	// ============ Common varaibles ==============================
	bAxisMoved						:		BOOL;						// History variable to save if axis has moved marker
	fbTriggerResetStart				:		R_TRIG;						// To diagnose rising edge of starting reset
	fbTriggerStartingStart			:		R_TRIG;						// To diagnose rising edge of starting start
END_VAR

// ===========================================================================
;
// ===========================================================================

PROPERTY bState_HaltDone : BOOL
GET
bState_HaltDone := bHaltDone;
END_GET
END_PROPERTY

PROPERTY bState_ResetDone : BOOL
GET
bState_ResetDone := bResetDone;
END_GET
END_PROPERTY

PROPERTY bState_StartingDone : BOOL
GET
bState_StartingDone := bStartingDone;
END_GET
END_PROPERTY

METHOD Enable
VAR_INPUT
	bComprAirEnable					:			BOOL;			// Enable of compressed air
	bAxisEnable						:			BOOL;			// Enable of axis
	bSensorEnable					:			BOOL;			// Enable of sensor
	bManualAxisEnable				:			BOOL;			// Enable manual axis control
END_VAR

VAR
	bManualEnable: BOOL;
END_VAR
	// Store inputs in local variables
	bCompresAirEnableLocal				:=				bComprAirEnable;
	bAxisEnableLocal					:=				bAxisEnable;
	bSensorEnableLocal					:=				bSensorEnable;
	bManualAxisEnableLocal				:=				bManualAxisEnable;
	
	// Axis enable
	fbAxis.Enable(bEnable				:=				bAxisEnableLocal);
	
	// Cylinder manual control enable 
	bManualCylinderEnableLocal			:=				bManualAxisEnableLocal		AND		bCompresAirEnableLocal;
	
	// Control buttons (enable Signal Handling)
	fbButtonAxisFw.Enable(bEnable		:=				bManualAxisEnableLocal		AND NOT fbButtonAxisBw.bOutputSignal);
	fbButtonAxisBw.Enable(bEnable		:=				bManualAxisEnableLocal		AND NOT fbButtonAxisFw.bOutputSignal);
END_METHOD

PROPERTY fAxisVelocity : LREAL
GET
fAxisVelocity := fAxisVelo;
END_GET
SET
fAxisVelo := fAxisVelocity;
END_SET
END_PROPERTY

METHOD Halt : BOOL
VAR_INPUT
	bHalt				:			BOOL;				// True if machine is in STATE ABORTING or STOPPING
END_VAR
	// Store halt request
	bHaltRequest				:=		bHalt;
	
	// Axis halt
	fbAxis.Halt(bDriveHalt		:=		bHaltRequest);
	
	// Setting halt state from axis feedback
	bHaltDone					:=		fbAxis.bState_HaltDone;
END_METHOD

METHOD InputOutput
VAR_INPUT
END_VAR
	// Axis buttons and output variables for axis
	fbButtonAxisFw.SetOutput();
	fbButtonAxisBw.SetOutput();

	bAxisError							:=					fbAxis.bError;
	nAxisErrorID						:=					fbAxis.nErrorID;
	bAxisMoves							:=					fbAxis.bMoving;
	
	fbButtonAxisFw.bInputSignal			:=					bButtonAxisFwIn;
	fbButtonAxisBw.bInputSignal			:=					bButtonAxisBwIn;
	bButtonAxisFwOut					:=					fbButtonAxisFw.bOutputSignal;
	bButtonAxisBwOut					:=					fbButtonAxisBw.bOutputSignal;
END_METHOD

METHOD Manual
VAR_INPUT
END_VAR

	IF fbButtonAxisFw.bOutputSignal THEN
		IF bHaltDone THEN
			bHaltDone	:=		FALSE;
		END_IF
		
		IF NOT bAxisMoved THEN
			bAxisMoved 	:=		TRUE;
		END_IF
		
		fbAxis.MoveFw();
		
	ELSIF fbButtonAxisBw.bOutputSignal THEN
		IF bHaltDone THEN
			bHaltDone	:=		FALSE;
		END_IF
		
		IF NOT bAxisMoved THEN
			bAxisMoved 	:=		TRUE;
		END_IF
	
		fbAxis.MoveBw();
	
	// No button is pressed and Halt is not done
	ELSIF NOT bHaltDone	THEN
		IF bAxisMoved THEN
			Halt(bHalt	:=	TRUE);
		END_IF
	
	// Halt done, but still requested
	ELSIF bHaltRequest THEN
		Halt(bHalt		:=	FALSE);
		
		bAxisMoved	:=	FALSE;
	END_IF
END_METHOD

METHOD Reset
VAR_INPUT
	bReset				:			BOOL;			// True if machine is in state RESETTING
END_VAR

	// Store reset request
	bResetRequest					:=			bReset;
	
	bAxisMoved						:=			FALSE;
	bHaltRequest					:=			FALSE;
	bHaltDone						:=			FALSE;
	
	// Trigger for resetting extending FBs 
	fbTriggerResetStart(CLK			:=			bReset);
	
	// Resetting axis
	fbAxis.Reset(bDriveReset		:=			bReset);
	
	bResetDone						:=			fbAxis.bState_ResetDone;
END_METHOD

METHOD Starting
VAR_INPUT
	bStarting					:				BOOL;			// True if machine is in state STARTING
END_VAR

	fbTriggerStartingStart(CLK			:=			bStarting);
	
	IF fbTriggerStartingStart.Q THEN
		bStartingDone					:=			FALSE;
	// Set axis velocity through axis property
		fbAxis.fTargetVelocity			:=			fAxisVelo;

	END_IF
	
	// Axis feedback from MC_Power of axis method Enable()
	IF fbAxis.bState_Enable THEN
		bStartingDone					:=			TRUE;
	END_IF
END_METHOD

METHOD Stop : BOOL
VAR_INPUT
	bStop					:				BOOL;				// True if machine is in state ABORTING or STOPPING
END_VAR
	// Store halt request
	bHaltRequest					:=				bStop;
	
	// Axis halt
	fbAxis.Stop(bDriveStop			:=				bHaltRequest);
	
	// Setting halt state from axis feedback
	bHaltDone						:=				fbAxis.bState_HaltDone;
END_METHOD

END_FUNCTION_BLOCK

// ---- 02_Subsystems/FB_SortingModule.TcPOU
FUNCTION_BLOCK FB_SortingModule EXTENDS FB_SubsystemRoot
VAR_INPUT
	bButtonCylMoveToWorkIn										:						BOOL;
	bButtonCylMoveToBaseIn										:						BOOL;
END_VAR
VAR_OUTPUT
	bCylError													:						BOOL;
	sCylErrorMsg												:						STRING;
	
	a_Temps														:						ARRAY [1..100] OF LREAL;
	
	bButtonCylMoveToWorkOut										:						BOOL;
	bButtonCylMoveToBaseOut										:						BOOL;
END_VAR
VAR
	bSorted														:						BOOL;								// Part picked at sorting module
	// Sensor with delay functionality
	fbSensorDelay												:						FB_SignalHandlingDelay;
	
	// Function block instance for cylinder
	fbCylinder													:						FB_CylinderBase;
	fbCylinderDiag												:						FB_CylinderDiag;
	fbCylinderTemp												:						FB_CylinderTemp;
	fbCylinderTempDiag											:						FB_CylinderTempDiag;
	fbCylinderTempRec											:						FB_CylinderTempRecord;
	// Interface instance for cylinder
	itfCylinder													:						I_Cylinder;
	// Time parameters for submodules
	tTimeOutCylinder											:						TIME;								// For cylinder with position diagnosis: time in which the cylinder shcould reach work / base position
	tTimeIntervalCylinder										:						TIME;								// Time of intervals to record the temperature of cylinder
	tSensorDelay												:						TIME;								// Sensor delay
	tMoveAxisDelay												:						TIME;								// Time delay to stop running axis
	// ========================== Temperature parameters for cylinder  ======================================================================
	nTempMinCyl													:						LREAL;								// For cylinder with temperature diagnosis: minimal temperature
	nTempMaxCyl													:						LREAL;								// For cylinder with temperature diagnosis: maximal temperature
	// Manual cylinder controll
	fbButtonCylMoveToWork										:						FB_SignalHandlingIntern;			// Button to move cylinder manually to work position
	fbButtonCylMoveToBase										:						FB_SignalHandlingIntern;			// Button to move cylinder manually to base position
	// Common variables
	fbTimerAxis													:						TON;								// Timer to run axis for certain amount of time
	fbTriggerCylAtWorkPos										:						R_TRIG;								// Trigger to recognize rising edge of cylinder being at work position
	eStateAutoAxis												:						E_StateSortingAutoAxis;				// State variable for automatic / semi-auto mode for axis movement
	eStateAutoCylinder											:						E_StateSortingAutoCylinder;			// State variable for automatic / semi-auto mode for cylinder movement
END_VAR

METHOD Automatic
VAR_INPUT
END_VAR
	fbTriggerCylAtWorkPos(		CLK			:=		itfCylinder.bState_AtWorkPos);

	CASE eStateAutoAxis OF
		
		E_StateSortingAutoAxis.WaitForCylinderAtWorkPos:
			IF fbTriggerCylAtWorkPos.Q THEN
				fbTimerAxis(	IN			:=		TRUE,
								PT			:=		tMoveAxisDelay);
				
				eStateAutoAxis				:=		E_StateSortingAutoAxis.MoveAxis;
			END_IF
		
		E_StateSortingAutoAxis.MoveAxis:
			fbTimerAxis();
			IF bHaltRequest THEN
				
				eStateAutoAxis				:=		E_StateSortingAutoAxis.StopAxis;
			ELSIF fbTimerAxis.Q THEN
				fbTimerAxis(	IN			:=		FALSE);
				
				bSorted						:=		TRUE;
			
				eStateAutoAxis				:=		E_StateSortingAutoAxis.StopAxis;
			ELSE
				fbAxis.MoveFw();
			END_IF
		
		E_StateSortingAutoAxis.StopAxis:
				bSorted						:=		FALSE;
				
				IF NOT bHaltDone THEN
					Stop(	bStop			:=		TRUE);
				ELSE	
					Stop(	bStop			:=		FALSE);
					eStateAutoAxis			:=		E_StateSortingAutoAxis.WaitForCylinderAtWorkPos;
				END_IF   
	END_CASE
	
	CASE eStateAutoCylinder OF
		E_StateSortingAutoCylinder.BoxDetected:
		
			itfCylinder.MoveToBase();
			
			IF fbSensorDelay.bOutputSignal THEN
				eStateAutoCylinder			:=		E_StateSortingAutoCylinder.MoveCylToWorkPos;	
			END_IF
				
		E_StateSortingAutoCylinder.MoveCylToWorkPos:
		
			itfCylinder.MoveToWork();
			
			IF itfCylinder.bState_AtWorkPos THEN
				eStateAutoCylinder			:=		E_StateSortingAutoCylinder.MoveCylToBasePos;
			END_IF
			
		E_StateSortingAutoCylinder.MoveCylToBasePos:
			itfCylinder.MoveToBase();
			
			IF itfCylinder.bState_AtBasePos THEN
				eStateAutoCylinder			:=		E_StateSortingAutoCylinder.BoxDetected;
			END_IF	
	END_CASE
END_METHOD

PROPERTY bState_CylAtBasePos : BOOL
GET
bState_CylAtBasePos			:=		itfCylinder.bState_AtBasePos;
END_GET
END_PROPERTY

PROPERTY bState_CylAtWorkPos : BOOL
GET
bState_CylAtWorkPos			:=		itfCylinder.bState_AtWorkPos;
END_GET
END_PROPERTY

METHOD CylinderOptions
VAR_INPUT
	bCylDiag							:				BOOL;						// If TRUE cylinder has diagnostic functionality
	bCylTemp							:				BOOL;						// If TRUE cylinder has temperature functionality
	bCylRecord							:				BOOL;						// If TRUE cylinder has record functionality
END_VAR

	IF 	bCylDiag THEN
		IF bCylTemp THEN
			fbCylinderTempDiag.fTempMin				:=			nTempMinCyl;
			fbCylinderTempDiag.fTempMax				:=			nTempMaxCyl;
			bCylError								:=			fbCylinderTempDiag.bError;
			sCylErrorMsg							:=			fbCylinderTempDiag.sErrorMsg;
				itfCylinder								:=			fbCylinderTempDiag;
		ELSE
			bCylError								:=			fbCylinderDiag.bError;
			sCylErrorMsg							:=			fbCylinderDiag.sErrorMsg;
			fbCylinderDiag.nTimeOut					:=			tTimeOutCylinder;			
				itfCylinder								:=			fbCylinderDiag;
		END_IF
	ELSE
		bCylError									:=			FALSE;
		sCylErrorMsg								:=			'';
		
		IF 	bCylTemp THEN
			IF bCylRecord THEN
				fbCylinderTempRec.nTimeInterval		:=			tTimeIntervalCylinder;
				fbCylinderTempRec.bRecordStart		:=			bCompresAirEnableLocal;
				
				fbCylinderTempRec.Record();
				
				a_Temps								:=			fbCylinderTempRec.aRecords;
				
					itfCylinder	:= fbCylinderTempRec;
			
			ELSE
					itfCylinder	:=	fbCylinderTemp;
			END_IF
		ELSE
					itfCylinder	:= fbCylinder;
		END_IF
			
	END_IF
	
	;
END_METHOD

METHOD Enable
VAR_INPUT
	bComprAirEnable					:			BOOL;			// Enable of compressed air
	bAxisEnable						:			BOOL;			// Enable of axis
	bSensorEnable					:			BOOL;			// Enable of sensor
	bManualAxisEnable				:			BOOL;			// Enable manual axis control
END_VAR

VAR
	bManualEnable: BOOL;
END_VAR

	SUPER^.Enable(	bComprAirEnable				:=	bComprAirEnable,
					bAxisEnable					:=	bAxisEnable,
					bSensorEnable				:=	bSensorEnable,
					bManualAxisEnable			:=	bManualAxisEnable);
					
	fbSensorDelay.Enable(bEnable				:=	bSensorEnable);
	
	fbButtonCylMoveToWork.Enable(bEnable		:=	bManualCylinderEnableLocal AND NOT itfCylinder.bState_AtWorkPos);					// bManualAxisEnableLocal AND bComprAirEnabledLocal	
	fbButtonCylMoveToBase.Enable(bEnable		:=	bManualCylinderEnableLocal AND NOT itfCylinder.bState_AtBasePos);					// bManualAxisEnableLocal AND bComprAirEnabledLocal
	
	fbButtonCylMoveToWork.bInputSignal			:=	NOT fbButtonCylMoveToBase.bInputSignal;
END_METHOD

METHOD InputOutput
VAR_INPUT
END_VAR

	SUPER^.InputOutput();
	
	fbSensorDelay.SetOutput();
	
	
	
	fbButtonCylMoveToWork.SetOutput();
	fbButtonCylMoveToBase.SetOutput();
	
	fbButtonCylMoveToWork.bInputSignal					:=		bButtonCylMoveToWorkIn;
	fbButtonCylMoveToBase.bInputSignal					:=		bButtonCylMoveToBaseIn;
	
	bButtonCylMoveToWorkOut								:=		fbButtonCylMoveToWork.bOutputSignal;
	bButtonCylMoveToBaseOut								:=		fbButtonCylMoveToBase.bOutputSignal;
END_METHOD

METHOD Maintenance
VAR_INPUT
END_VAR

	THIS^.Manual();
END_METHOD

METHOD Manual
VAR_INPUT
END_VAR
	
	SUPER^.Manual();
	
	IF fbButtonCylMoveToWork.bOutputSignal THEN
		itfCylinder.MoveToWork();
	ELSIF	fbButtonCylMoveToBase.bOutputSignal THEN
		itfCylinder.MoveToBase();
	END_IF
END_METHOD

PROPERTY nProp_CylTempMax : LREAL
GET
nProp_CylTempMax		:=		nTempMaxCyl;
END_GET
SET
nTempMaxCyl			:=		nProp_CylTempMax;
END_SET
END_PROPERTY

PROPERTY nProp_CylTempMin : LREAL
GET
nProp_CylTempMin		:=		nTempMinCyl;
END_GET
SET
nTempMinCyl			:=		nProp_CylTempMin;
END_SET
END_PROPERTY

METHOD Reset
VAR_INPUT
	bReset				:			BOOL;			// True if machine is in state RESETTING
END_VAR

	SUPER^.Reset(	bReset			:=			bReset);
	
	IF fbTriggerResetStart.Q THEN
	
	fbTimerAxis(	IN				:=			FALSE);			
	
	itfCylinder.Reset();
	
	END_IF
END_METHOD

METHOD ResetState
VAR_INPUT
END_VAR
// =========================================================
	eStateAutoAxis					:=			E_StateSortingAutoAxis.WaitForCylinderAtWorkPos;
	eStateAutoCylinder				:=			E_StateSortingAutoCylinder.BoxDetected;
// =========================================================
END_METHOD

METHOD Semiautomatic
VAR_INPUT
END_VAR
	
	THIS^.Automatic();
END_METHOD

METHOD Starting
VAR_INPUT
	bStarting					:				BOOL;			// True if machine is in state STARTING
END_VAR

	SUPER^.Starting(	bStarting			:=			bStarting);
	
	fbSensorDelay.tDelay					:=			tSensorDelay;
END_METHOD

PROPERTY tProp_AxisMoving : TIME
GET
tProp_AxisMoving		:=		tMoveAxisDelay;
END_GET
SET
tMoveAxisDelay			:=		tProp_AxisMoving;
END_SET
END_PROPERTY

PROPERTY tProp_CylRecInterval : TIME
GET
tProp_CylRecInterval		:=			tTimeIntervalCylinder;
END_GET
SET
tTimeIntervalCylinder			:=			tProp_CylRecInterval;
END_SET
END_PROPERTY

PROPERTY tProp_CylTimeOut : TIME
GET
tProp_CylTimeOut			:=			tTimeOutCylinder;
END_GET
SET
tTimeOutCylinder		:=			tProp_CylTimeOut;
END_SET
END_PROPERTY

PROPERTY tProp_SensorDelay : TIME
GET
tProp_SensorDelay			:=			fbSensorDelay;
END_GET
SET
fbSensorDelay			:=			tProp_SensorDelay;
END_SET
END_PROPERTY

END_FUNCTION_BLOCK

// ---- 03_Machine/FB_Machine.TcPOU
FUNCTION_BLOCK FB_Machine
VAR_INPUT
	// ========================== SEPARATING MODULE =======================================
	// Separating module - clamp cylinder
	bSeparatingClampDiag						:		BOOL	:=	FALSE;
	bSeparatingClampTemp						:		BOOL	:=	TRUE;
	bSeparatingClampRecord						:		BOOL	:=	TRUE;
	// Separating module - barrier cylinder
	bSeparatingBarrierDiag						:		BOOL	:=	TRUE;
	bSeparatingBarrierTemp						:		BOOL	:=	TRUE;
	bSeparatingBarrierRecord					:		BOOL	:=	FALSE;
	// ========================== SORTING MODULES ==========================================
	bMetalSortingCylinderDiag					:		BOOL	:= 	TRUE;
	bMetalSortingCylinderTemp					:		BOOL	:=	FALSE;
	bMetalSortingCylinderRecord					:		BOOL	:=	FALSE;
	
	bPlasticSortingCylinderDiag					:		BOOL	:=	FALSE;
	bPlasticSortingCylinderTemp					:		BOOL	:=	FALSE;
	bPlasticSortingCylinderRecord				:		BOOL	:=	FALSE;
END_VAR
VAR
	// ============================= ERROR ==================================================
	bError										:		BOOL;
	// ========================== Axis Variable =============================================
	fAxisVelo									:		LREAL;
	fAxisVeloLastCycle							:		LREAL;
	// ======================== State machine variables =====================================
	bStarted									:		BOOL;
	bStopped									:		BOOL;
	bReset								AT %Q* 	: 		BOOL;
	bAborted									:		BOOL;
	bIdle										:		BOOL;
	bAuto										:		BOOL;
	bSemi										:		BOOL;
	bManual										:		BOOL;
	bMaintenance								:		BOOL;
	// ========================== Machine submodules ========================================
	fbSeparatingModule							:		FB_SeparatingModule;
	fbMetalSortingModule						:		FB_SortingModule;
	fbPlasticSortingModule						:		FB_SortingModule;
	fbComprAir									:		FB_SignalHandlingIntern;
	fbPowerSupply								:		FB_SignalHandlingIntern;
	// Visualization
	// ========================== Buttons ========================================
	fbButtonStart								:		FB_SignalHandlingIntern;
	fbButtonStop								:		FB_SignalHandlingIntern;
	fbButtonReset								:		FB_SignalHandlingIntern;
	fbButtonAbort								:		FB_SignalHandlingIntern;
	fbButtonAuto								:		FB_SignalHandlingIntern;
	fbButtonSemi								:		FB_SignalHandlingIntern;
	fbButtonManual								:		FB_SignalHandlingIntern;
	fbButtonMaintenance							:		FB_SignalHandlingIntern;
	fbButtonComprAir							:		FB_SignalHandlingIntern;
	fbButtonPower								:		FB_SignalHandlingIntern;
	// ========================== State machine ==================================
	fbStateMachineAuto							:		PS_PackML_StateMachine_Auto;
	fbStateMachineSemiAuto						:		PS_PackML_StateMachine_SemiAuto;
	fbStateMachineManual						:		PS_PackML_StateMachine_Manual;
	fbStateMachineMaintenance					:		PS_PackML_StateMachine_Maintenance;
	
	e_PMLState									:		E_PMLState			:=	E_PMLState.IDLE;
	e_PMLStateRequest							:		E_PMLState;
	e_PMLUnitMode								:		E_PMLUnitMode		:=	E_PMLUnitMode.IDLE;
	e_PMLUnitModeRequest						:		E_PMLUnitMode;
	// fbUnitModeManager
	// ======================= Common variables ===================================
	bInit										:		BOOL;
	bAxisEnable									:		BOOL;
	bManualAxisEnable							:		BOOL;
	
	fbTriggerStartButton						:		R_TRIG;
	
	nBoxesOnTransport							:		UINT;
	
	aClampTemps									:		ARRAY [1..100] OF LREAL;
	aBarrierTemps								:		ARRAY [1..100] OF LREAL;
	aMetalCylTemps								:		ARRAY [1..100] OF LREAL;
	aPlasticCylTemps							:		ARRAY [1..100] OF LREAL;
END_VAR
VAR CONSTANT
	// ======================= Axis parameters ===================================
	nAxisVeloAutomatic							:		LREAL	:=		100.0;
	nAxisVeloNonAutomatic						:		LREAL	:=		50.0;
	// =============== Separating module parameters ===============================
	tSeparatingTimeOutClamp						:		TIME	:=		T#4S;
	tSeparatingRecordIntervalClamp				:		TIME	:=		T#1S;
	
	tSeparatingTimeOutBarrier					:		TIME	:=		T#3S;
	tSeparatingRecordIntervalBarrier			:		TIME	:=		T#1S;
	tSeparatingTimeBarrierAtWork				:		TIME	:=		T#3.5S;
	// =============== Sorting module parameters ==================================
	tSortingMetalTimeOutCyl						:		TIME	:=		T#3S;
	tSortingMetalRecordIntervalCyl				:		TIME	:=		T#1S;
	tSortingMetalSensorDelay					:		TIME	:=		T#2S;
	tSortingMetalMoveAxisDelay					:		TIME	:=		T#3S;

	tSortingPlasticTimeOutCyl					:		TIME	:=		T#3S;
	tSortingPlasticRecordIntervalCyl			:		TIME	:=		T#1S;
	tSortingPlasticSensorDelay					:		TIME	:=		T#2S;
	tSortingPlasticMoveAxisDelay				:		TIME	:=		T#3S;
END_VAR

END_FUNCTION_BLOCK
